# EPICS substitutions: tds3000App/Db/tds.substitutions
file tdsChan.template{
  {N=1}
  {N=2}
  {N=3}
  {N=4}
}
